{attribute 'qualified_only'}
{attribute 'to_string'}
TYPE E_GROUP_CHECK :
(
  CHECK_NULL,
  CHECK_GROUP_REF_INVALID := 10,
  CHECK_AXIS_REF_INVALID,
  CHECK_CTRL_INVALID,
  CHECK_STATE_INVALID,
  CHECK_Mover_ITF_REF_INVALID,
  CHECK_XPU_INFO_REF_INVALID,


  CHECK_ERROR             :=  9000,
  CHECK_DONE              := 10000
)UINT;
END_TYPE

(* stored: Version 1.1.0.1
   DUT E_GROUP_CHECK: Id {657a9c8a-03bc-41ac-a86a-300e2f865fd1} *)
